FUNCTION_BLOCK LINX215_LWEB (* Service Interface Function Block Type *)
  (* Standard: 61499-2 *)
  (* Version 0.0, 3/14/2024, linkwise-linn, LOYTEC electronics GmbH, template *)
  PACKAGE Main;
  (* Compiler Cpp LOYTEC electronics GmbH builtin 1.0 *)
  {SET_ATTRIBUTE(Configuration.FBType.DPAL.SFBLWEB, )}
  {SET_ATTRIBUTE(Runtime.FBType.ImplementingType, Loytec.DPAL#DYNGEN_DPALSFB)}
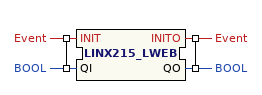
  EVENT_INPUT
    INIT WITH QI;
  END_EVENT
  EVENT_OUTPUT
    INITO WITH QO;
  END_EVENT
  VAR_INPUT
    QI : BOOL;
  END_VAR
  VAR_OUTPUT
    QO : BOOL;
  END_VAR
  SERVICE APPLICATION/RESOURCE
    SEQUENCE 
    END_SEQUENCE
  END_SERVICE
END_FUNCTION_BLOCK
